// TIA Portal V17 export
// export: Created 2024-09-02T12:50:19.6078163Z, ExportSetting WithDefaults, DisplayName Totally Integrated Automation Portal, DisplayVersion V17, DisplayName TIA Portal Openness, DisplayVersion V17, DisplayName TIA Portal Version Control Interface, DisplayVersion V17, DisplayName STEP 7 Professional, DisplayVersion V17, DisplayName STEP 7 Safety, DisplayVersion V17, DisplayName WinCC Professional, DisplayVersion V17
DATA_BLOCK "AnwDB_Omron_OP70_2"   // DB190
{ S7_Optimized_Access := 'FALSE'; DB_Accessible_From_OPC_UA := 'FALSE' }
VERSION : 0.1
// stored: AutoNumber false, DBAccessibleFromOPCUA false, IsOnlyStoredInLoadMemory false, IsWriteProtectedInAS false
   VAR
      Output : Struct
         Ready : Bool;
         Busy : Bool;
         Done : Bool;
         Ok : Bool;
         NOK : Bool;
         Error : Bool;
         ErrorCode : Bool;
         Data : Array[0..7] of DWord;
      END_STRUCT;
      Input : Struct
         Restart_Result : Bool;
         Ack_Active : Bool;
         Trigger : Bool;
      END_STRUCT;
      HMI : Struct
         Button : Struct
            Lighting : Struct
               Layout : Int;
               active : Bool;
            END_STRUCT;
            Read : Struct
               Layout : Int;
               active : Bool;
            END_STRUCT;
            Reset : Struct
               Layout : Int;
               active : Bool;
            END_STRUCT;
         END_STRUCT;
         Status : Struct
            Input : Struct
               Restart_Result : Bool;
               Ack_Active : Bool;
               Trigger : Bool;
            END_STRUCT;
            Output : Struct
               Ready : Bool;
               Busy : Bool;
               Done : Bool;
               Ok : Bool;
               NOK : Bool;
               Error : Bool;
               ErrorCode : Bool;
               Data : Array[0..7] of DWord;
            END_STRUCT;
            Result : Struct
               Damper_OP50_1 : Bool;
               Damper_OP50_2 : Bool;
               Damper_OP50_3 : Bool;
               Filter_OP60 : Bool;
               Ball_OP70_1 : Bool;
               Damper_OP70_1 : Bool;
               Dowel_1_OP60 : Bool;
               Dowel_2_OP60 : Bool;
            END_STRUCT;
         END_STRUCT;
      END_STRUCT;
   END_VAR
BEGIN
END_DATA_BLOCK
